FUNCTION_BLOCK PalletizerElevator EXTENDS Elevator
VAR_INPUT
END_VAR
VAR_OUTPUT
	isMoving : BOOL;
END_VAR
VAR
	fbElevatorMoving : Sensor;
	fbElevatorUp : BoolOut;
	fbElevatorDown : BoolOut;
	fbElevatorTopLimit : BoolOut;
	fbElevatorBottomLimit : BoolOut;
END_VAR

super^();
isMoving := fbElevatorMoving.bSignal;

METHOD  executeCmd : BOOL
VAR_INPUT
	
END_VAR
CASE eCmd OF
	eUP:
		moveUp();
	eDOWN:
		moveDown();
	eUP_TO_LIMIT:
		moveTopLimit();
	eDOWN_TO_LIMIT:
		moveBottomLimit();
END_CASE
END_METHOD

PROPERTY getElevatorMoving : I_StepCondition
GET
getElevatorMoving := fbElevatorMoving.getSignal;
END_GET
END_PROPERTY

METHOD moveBottomLimit : BOOL
VAR_INPUT
END_VAR
fbElevatorDown.setValue := FALSE;
fbElevatorUp.setValue := FALSE;

fbElevatorTopLimit.setValue := FALSE;
fbElevatorBottomLimit.setValue := TRUE;
END_METHOD

METHOD moveDown : BOOL
VAR_INPUT
END_VAR
fbElevatorDown.setValue := TRUE;
fbElevatorUp.setValue := FALSE;

fbElevatorTopLimit.setValue := FALSE;
fbElevatorBottomLimit.setValue := FALSE;
END_METHOD

METHOD moveTopLimit : BOOL
VAR_INPUT
END_VAR
fbElevatorDown.setValue := FALSE;
fbElevatorUp.setValue := FALSE;

fbElevatorTopLimit.setValue := TRUE;
fbElevatorBottomLimit.setValue := FALSE;
END_METHOD

METHOD moveUp : BOOL
VAR_INPUT
END_VAR
fbElevatorUp.setValue := TRUE;
fbElevatorDown.setValue := FALSE;

fbElevatorTopLimit.setValue := FALSE;
fbElevatorBottomLimit.setValue := FALSE;
END_METHOD

END_FUNCTION_BLOCK

(* stored: Version 1.1.0.1, ProductVersion 3.1.4024.2
   POU PalletizerElevator: Id {bd2ea0f4-c169-461a-88aa-19be27edaaa5}, SpecialFunc None
   Method executeCmd: Id {bcaee20d-1518-461c-a9ba-abd0cf16fc6a}
   Property getElevatorMoving: Id {59fab772-9080-4a6d-8461-0b473e1c1552}
   Get Get: Id {afbe618a-6e76-4617-8d5d-ebb798925f13}
   Method moveBottomLimit: Id {920b6b28-efc3-411e-a8ec-d1f8b52cfdb5}
   Method moveDown: Id {73b801bf-e72e-41ab-ac7b-579ada3843c5}
   Method moveTopLimit: Id {a02f38fd-3a51-4986-a492-336f2cc6a774}
   Method moveUp: Id {c7f781fc-6698-47a1-8530-f8c7485ab296} *)
